(* PLC project HydMotion Functions library, Porcheson Hydraulic Motion 0.0 *)
(* stored: creationDateTime 2023-02-10T00:00:00, modificationDateTime 2026-02-10T00:00:00 *)

TYPE HYD_AxisMotion : STRUCT
  SEGMENTTAG : USINT;
  SEGMENTTYPE : USINT;
  PLANNER : USINT;
  MODE : USINT;
  ENDCONDITION : USINT;
  DIRECTION : USINT;
  SETPOSITION : REAL;
  SETVELOCITY : REAL;  (* 仅在速度/流量控制模式下使用，表示目标速度； *)
  SETFLOW : REAL;  (* 仅在速度/流量控制模式下使用，表示目标流量；在位置控制模式下忽略 *)
  SETPRESSURE : REAL;
  ACCELERATION : REAL;
  DECELERATION : REAL;
  DURATION : REAL;
  PRESSURERAMPRATE : REAL;
  ACTPOSITION : REAL;
  ACTVELOCITY : REAL;
  ACTFLOW : REAL;
  ACTPRESSURE : REAL;
  TIMESTAMP : REAL;
END_STRUCT;
END_TYPE

FUNCTION_BLOCK HYD_MoveProfile
  VAR_INPUT
    AXISID : SINT;
    EXECUTE : BOOL;
    MOTION : HYD_AxisMotion;
    BUFFERMODE : INT;
  END_VAR
  VAR_OUTPUT
    DONE : BOOL;
    BUSY : BOOL;
    ACTIVE : BOOL;
    COMMANDABORTED : BOOL;
    ERROR : BOOL;
    ERRORID : WORD;
  END_VAR
  VAR
    Execute0 : BOOL;
    Done0 : BOOL;
    Active0 : BOOL;
    _PENDING : BOOL;
    _EXEC_ID : WORD;
  END_VAR

 {{ extern void __mcl_cmd_MoveProfile(HYD_MOVEPROFILE *data__);	__mcl_cmd_MoveProfile(data__);	 }}			
END_FUNCTION_BLOCK

FUNCTION_BLOCK HYD_LoadProfile
  VAR_INPUT
    AXISID : SINT;
    EXECUTE : BOOL;
    MOTION : HYD_AxisMotion;
  END_VAR
  VAR_OUTPUT
    DONE : BOOL;
    BUSY : BOOL;
    ERROR : BOOL;
    ERRORID : WORD;
  END_VAR
  VAR
    Execute0 : BOOL;
    Done0 : BOOL;
  END_VAR

						{{ extern void __mcl_cmd_LoadProfile(HYD_LOADPROFILE *data__);	__mcl_cmd_LoadProfile(data__);	 }}	
					
END_FUNCTION_BLOCK

FUNCTION_BLOCK HYD_Stop
  VAR_INPUT
    AXISID : SINT;
    EXECUTE : BOOL;
    DECELERATION : REAL;
  END_VAR
  VAR_OUTPUT
    DONE : BOOL;
    BUSY : BOOL;
    COMMANDABORTED : BOOL;
    ERROR : BOOL;
    ERRORID : WORD;
  END_VAR
  VAR
    Execute0 : BOOL;
    Done0 : BOOL;
    Active0 : BOOL;
    _PENDING : BOOL;
  END_VAR

						{{ extern void __mcl_cmd_Stop(HYD_STOP *data__);	__mcl_cmd_Stop(data__);	 }}	
					
END_FUNCTION_BLOCK

FUNCTION_BLOCK HYD_Hold
  VAR_INPUT
    AXISID : SINT;
    EXECUTE : BOOL;
  END_VAR
  VAR_OUTPUT
    DONE : BOOL;
    BUSY : BOOL;
    ERROR : BOOL;
    ERRORID : WORD;
  END_VAR
  VAR
    EXECUTE0 : BOOL;
    DONE0 : BOOL;
    _PENDING : BOOL;
  END_VAR

{{ extern void __mcl_cmd_Hold(HYD_HOLD*); __mcl_cmd_Hold(data__); }} 
END_FUNCTION_BLOCK

FUNCTION_BLOCK HYD_Resume
  VAR_INPUT
    AXISID : SINT;
    EXECUTE : BOOL;
  END_VAR
  VAR_OUTPUT
    DONE : BOOL;
    BUSY : BOOL;
    ERROR : BOOL;
    ERRORID : WORD;
  END_VAR
  VAR
    EXECUTE0 : BOOL;
    DONE0 : BOOL;
    _PENDING : BOOL;
  END_VAR

{{ extern void __mcl_cmd_Resume(HYD_RESUME*); __mcl_cmd_Resume(data__); }} 
END_FUNCTION_BLOCK

(* This Function Block commands a controlled motion to a specified absolute position. *)
FUNCTION_BLOCK HYD_MoveAbsolute
  VAR_INPUT
    AXISID : SINT;
    EXECUTE : BOOL;
    CONTINUOUSUPDATE : BOOL;
    POSITION : REAL;
    VELOCITY : REAL;
    ACCELERATION : REAL;
    DECELERATION : REAL;
    JERK : REAL;
    DIRECTION : SINT;
    BUFFERMODE : INT;
  END_VAR
  VAR_OUTPUT
    DONE : BOOL;
    BUSY : BOOL;
    ACTIVE : BOOL;
    COMMANDABORTED : BOOL;
    ERROR : BOOL;
    ERRORID : WORD;
  END_VAR
  VAR
    EXECUTE0 : BOOL;
    DONE0 : BOOL;
    ACTIVE0 : BOOL;
    _PENDING : BOOL;
    _EXEC_ID : WORD;
  END_VAR

						{{ extern void __mcl_cmd_MoveAbsolute(HYD_MOVEABSOLUTE*); __mcl_cmd_MoveAbsolute(data__); }}	
					
END_FUNCTION_BLOCK

FUNCTION_BLOCK HYD_MoveContinuousAbsolute
  VAR_INPUT
    AXISID : SINT;
    EXECUTE : BOOL;
    POSITION : REAL;
    VELOCITY : REAL;
    ENDVELOCITY : REAL;
    ENDVELOCITYDIRECTION : SINT;
    ACCELERATION : REAL;
    DECELERATION : REAL;
    JERK : REAL;
    DIRECTION : SINT;
    ADAPTENDVELTOAVOIDOVERSHOOT : BOOL;
    PRESSURELIMIT : REAL;
  END_VAR
  VAR_OUTPUT
    INENDVELOCITY : BOOL;
    POSITIONREACHED : BOOL;
    BUSY : BOOL;
    COMMANDABORTED : BOOL;
    ERROR : BOOL;
    ERRORID : WORD;
  END_VAR
  VAR
    EXECUTE0 : BOOL;
    INENDVELOCITY0 : BOOL;
    POSITIONREACHED0 : BOOL;
    _PENDING : BOOL;
    _EXEC_ID : WORD;
  END_VAR

{{ extern void __mcl_cmd_MoveContinuousAbsolute(HYD_MOVECONTINUOUSABSOLUTE*); __mcl_cmd_MoveContinuousAbsolute(data__); }} 
END_FUNCTION_BLOCK

(* This Function Block commands a never ending controlled motion at a specified velocity. *)
FUNCTION_BLOCK HYD_MoveVelocity
  VAR_INPUT
    AXISID : SINT;
    EXECUTE : BOOL;
    CONTINUOUSUPDATE : BOOL;
    VELOCITY : REAL;
    ACCELERATION : REAL;
    DECELERATION : REAL;
    JERK : REAL;
    DIRECTION : SINT;
    BUFFERMODE : INT;
    PRESSURELIMIT : REAL;
  END_VAR
  VAR_OUTPUT
    INVELOCITY : BOOL;
    BUSY : BOOL;
    ACTIVE : BOOL;
    COMMANDABORTED : BOOL;
    ERROR : BOOL;
    ERRORID : WORD;
  END_VAR
  VAR
    EXECUTE0 : BOOL;
    INVELOCITY0 : BOOL;
    ACTIVE0 : BOOL;
    _PENDING : BOOL;
    _EXEC_ID : WORD;
  END_VAR

{{ extern void __mcl_cmd_MoveVelocity(HYD_MOVEVELOCITY*); __mcl_cmd_MoveVelocity(data__); }} 
END_FUNCTION_BLOCK

(* This Function Block makes the transition from the state ‘ErrorStop’ to ‘Disabled’ by resetting all internal axis-related errors *)
FUNCTION_BLOCK HYD_Reset
  VAR_INPUT
    AXISID : SINT;
    EXECUTE : BOOL;
  END_VAR
  VAR_OUTPUT
    DONE : BOOL;
    BUSY : BOOL;
    ERROR : BOOL;
    ERRORID : WORD;
  END_VAR
  VAR
    EXECUTE0 : BOOL;
    DONE0 : BOOL;
  END_VAR

{{ extern void __mcl_cmd_Reset(HYD_RESET*); __mcl_cmd_Reset(data__); }} 
END_FUNCTION_BLOCK

(* This Function Block commands pressure closed control. FLOWLIMITPERCENT is the pressure-segment flow cap as a percentage of 20 L/min; valid range is (0,100], default 100. *)
FUNCTION_BLOCK HYD_PressureHandle
  VAR_INPUT
    AXISID : SINT;
    EXECUTE : BOOL;
    CONTINUOUSUPDATE : BOOL;
    PRESSURE : REAL;
    PRESSURERAMPRATE : REAL;
    DURATION : REAL;
    FLOWLIMITPERCENT : REAL := 100;
    BUFFERMODE : INT;
  END_VAR
  VAR_OUTPUT
    INPRESSURE : BOOL;
    DONE : BOOL;
    BUSY : BOOL;
    ACTIVE : BOOL;
    COMMANDABORTED : BOOL;
    ERROR : BOOL;
    ERRORID : WORD;
  END_VAR
  VAR
    EXECUTE0 : BOOL;
    INPRESSURE0 : BOOL;
    ACTIVE0 : BOOL;
    _PENDING : BOOL;
    _EXEC_ID : WORD;
  END_VAR

{{ extern void __mcl_cmd_PressureHandle(HYD_PRESSUREHANDLE*); __mcl_cmd_PressureHandle(data__); }} 
END_FUNCTION_BLOCK

(* This allocates a simulation Axis, for testing.One axis per instanciated FB. *)
FUNCTION_BLOCK HYD_CreateMotion
  VAR_INPUT
    USE_RECIPE : BOOL := 0;
    FLOW_TO_PUMPSPEED : REAL := 20.0;
    PUMPSPEED_LIMIT : REAL := 1800.0;
    USE_SIMULATION : BOOL := 0;
    MECHANISM_TYPE : SINT := 0;
  END_VAR
  VAR_OUTPUT
    AXISID : SINT;
    DONE : BOOL;
    BUSY : BOOL;
    ERROR : BOOL;
    ERRORID : WORD;
  END_VAR
  VAR
    DONE0 : BOOL;
    _RESERVED_AXIS : SINT;
    _RESERVED_SLOT : USINT;
    _VALIDATION_TOKEN : USINT;
    _CREATE_ACTIVE : BOOL;
    _FRAMEWORK_GENERATION : WORD;
  END_VAR

						{{ extern void __mcl_cmd_CreateMotion(HYD_CREATEMOTION*); __mcl_cmd_CreateMotion(data__); }} 
					
END_FUNCTION_BLOCK

(* Atomically validates and commits five-point toggle geometry. *)
FUNCTION_BLOCK HYD_ConfigureToggleMechanism
  VAR_INPUT
    AXISID : SINT;
    EXECUTE : BOOL;
    LR : LREAL;
    LF : LREAL;
    LPF : LREAL;
    LPK : LREAL;
    LD : LREAL;
    HF : LREAL;
    HM : LREAL;
    DC : LREAL;
    SM : LREAL;
    XHANDOFF : LREAL;
    SIGMA_K : SINT;
    SIGN_B : SINT;
    TAU_S : SINT;
    SIGMA_C : SINT := -1;
  END_VAR
  VAR_OUTPUT
    DONE : BOOL;
    BUSY : BOOL;
    ERROR : BOOL;
    ERRORID : WORD;
    CONFIG_VERSION : WORD;
  END_VAR
  VAR
    EXECUTE0 : BOOL;
    VALIDATION_TOKEN : USINT;
    ACTIVE : BOOL;
    CONFIG_AXIS : SINT;
    _FRAMEWORK_GENERATION : WORD;
  END_VAR

{{ extern void __mcl_cmd_ConfigureToggleMechanism(HYD_CONFIGURETOGGLEMECHANISM*); __mcl_cmd_ConfigureToggleMechanism(data__); }} 
END_FUNCTION_BLOCK

(* Reads the committed five-point toggle geometry and safe envelope. *)
FUNCTION_BLOCK HYD_ReadToggleMechanism
  VAR_INPUT
    AXISID : SINT;
    ENABLE : BOOL;
  END_VAR
  VAR_OUTPUT
    VALID : BOOL;
    USING_DEFAULTS : BOOL;
    LR : LREAL;
    LF : LREAL;
    LPF : LREAL;
    LPK : LREAL;
    LD : LREAL;
    HF : LREAL;
    HM : LREAL;
    DC : LREAL;
    SM : LREAL;
    XHANDOFF : LREAL;
    SIGMA_K : SINT;
    SIGN_B : SINT;
    TAU_S : SINT;
    SIGMA_C : SINT;
    CONFIG_VERSION : WORD;
    X_GEOMETRY_MIN : LREAL;
    X_HANDOFF_EFFECTIVE : LREAL;
    XS_MIN : LREAL;
    XS_MAX : LREAL;
    K_MIN : LREAL;
    K_MAX : LREAL;
    ERROR : BOOL;
    ERRORID : WORD;
  END_VAR

{{ extern void __mcl_cmd_ReadToggleMechanism(HYD_READTOGGLEMECHANISM*); __mcl_cmd_ReadToggleMechanism(data__); }} 
END_FUNCTION_BLOCK

(* set feedback to motion. *)
FUNCTION_BLOCK HYD_SetAxisFeedback
  VAR_INPUT
    AXISID : SINT;
    ENABLE : BOOL;
    ACT_POSITION : REAL;
    ACT_VELOCITY : REAL;
    ACT_FLOW : REAL;
    ACT_PRESSURE : REAL;
    TIMESTAMP : REAL;
  END_VAR
  VAR_OUTPUT
    DONE : BOOL;
    BUSY : BOOL;
    ERROR : BOOL;
    ERRORID : WORD;
  END_VAR
  VAR
    DONE0 : BOOL;
  END_VAR

						{{ extern void __mcl_cmd_SetAxisFeedback(HYD_SETAXISFEEDBACK*); __mcl_cmd_SetAxisFeedback(data__); }} 
					
END_FUNCTION_BLOCK

(* write shared system-level pump feedback; one pump serves multiple axes. *)
FUNCTION_BLOCK HYD_SetPumpFeedback
  VAR_INPUT
    ENABLE : BOOL;
    PUMP_SPEED_RPM : REAL;
    PUMP_ANGLE_DEG : REAL;
    PUMP_TORQUE_PCT_TN : REAL;
    TIMESTAMP : REAL;
  END_VAR
  VAR_OUTPUT
    DONE : BOOL;
    BUSY : BOOL;
    ERROR : BOOL;
    ERRORID : WORD;
  END_VAR

{{ extern void __mcl_cmd_SetPumpFeedback(HYD_SETPUMPFEEDBACK*); __mcl_cmd_SetPumpFeedback(data__); }} 
END_FUNCTION_BLOCK

(* get only one pump speed command from motion. *)
FUNCTION_BLOCK HYD_GetPumpRequest
  VAR_INPUT
    ENABLE : BOOL;
    STRATEGY : SINT;
    ALLOW_NEGATIVE : BOOL;
  END_VAR
  VAR_OUTPUT
    PUMPSPEED : REAL;
    CONFLICT : BOOL;
    BUSY : BOOL;
    DONE : BOOL;
    ERROR : BOOL;
    ERRORID : WORD;
  END_VAR
  VAR
    DONE0 : BOOL;
  END_VAR

						{{ extern void __mcl_cmd_GetPumpRequest(HYD_GETPUMPREQUEST*); __mcl_cmd_GetPumpRequest(data__); }} 
					
END_FUNCTION_BLOCK

(* get axis status from motion. *)
FUNCTION_BLOCK HYD_ReadStatus
  VAR_INPUT
    AXISID : SINT;
    ENABLE : BOOL;
  END_VAR
  VAR_OUTPUT
    VALID : BOOL;
    BUSY : BOOL;
    ERROR : BOOL;
    ERRORID : WORD;
    STATE : UINT;
    PRESSURECONTROLLERAPPLIED : INT;
    MECHANISMTYPE : SINT;
    ACTUATORDIRECTION : SINT;
    ACTUATORPOSITION : REAL;
    ACTUATORVELOCITYCOMMAND : REAL;
    VELOCITYRATIO : REAL;
    MECHANISMCONFIGVERSION : WORD;
    REQUESTEDFLOW : REAL;
    MAXFLOW : REAL;
    MAXTEMPLATEVELOCITY : REAL;
    EFFECTIVECYLINDERGAIN : REAL;
    FLOWLIMITACTIVE : BOOL;
    PUMPSPEEDLIMITACTIVE : BOOL;
    PRESSURELIMITACTIVE : BOOL;
    SOFTLIMITACTIVE : BOOL;
    DERATED : BOOL;
  END_VAR

						{{ extern void __mcl_cmd_ReadStatus(HYD_READSTATUS*); __mcl_cmd_ReadStatus(data__); }} 
					
END_FUNCTION_BLOCK

(* get axis error from motion. *)
FUNCTION_BLOCK HYD_ReadError
  VAR_INPUT
    AXISID : SINT;
    ENABLE : BOOL;
  END_VAR
  VAR_OUTPUT
    VALID : BOOL;
    BUSY : BOOL;
    ERROR : BOOL;
    ERRORID : WORD;
  END_VAR

						{{ extern void __mcl_cmd_ReadError(HYD_READERROR*); __mcl_cmd_ReadError(data__); }} 
					
END_FUNCTION_BLOCK

(* get axis simfeedback from motion. *)
FUNCTION_BLOCK HYD_ReadSimFeedback
  VAR_INPUT
    AXISID : SINT;
    ENABLE : BOOL;
  END_VAR
  VAR_OUTPUT
    VALID : BOOL;
    BUSY : BOOL;
    ERROR : BOOL;
    ERRORID : WORD;
    POSITION : REAL;
    VELOCITY : REAL;
    FLOW : REAL;
    PRESSURE : REAL;
  END_VAR

						{{ extern void __mcl_cmd_ReadSimFeedback(HYD_READSIMFEEDBACK*); __mcl_cmd_ReadSimFeedback(data__); }} 
					
END_FUNCTION_BLOCK

FUNCTION_BLOCK HYD_ReadParameter
  VAR_INPUT
    AXISID : SINT;
    ENABLE : BOOL;
    PARAMETERNUMBER : INT;
  END_VAR
  VAR_OUTPUT
    VALID : BOOL;
    BUSY : BOOL;
    ERROR : BOOL;
    ERRORID : WORD;
    VALUE : LREAL;
  END_VAR
  VAR
    ENABLE0 : BOOL;
  END_VAR

{{ extern void __mcl_cmd_ReadParameter(HYD_READPARAMETER*); __mcl_cmd_ReadParameter(data__); }}
END_FUNCTION_BLOCK

FUNCTION_BLOCK HYD_WriteParameter
  VAR_INPUT
    AXISID : SINT;
    EXECUTE : BOOL;
    PARAMETERNUMBER : INT;
    VALUE : LREAL;
  END_VAR
  VAR_OUTPUT
    DONE : BOOL;
    BUSY : BOOL;
    ERROR : BOOL;
    ERRORID : WORD;
  END_VAR
  VAR
    EXECUTE0 : BOOL;
    DONE0 : BOOL;
  END_VAR

{{ extern void __mcl_cmd_WriteParameter(HYD_WRITEPARAMETER*); __mcl_cmd_WriteParameter(data__); }}
END_FUNCTION_BLOCK

FUNCTION_BLOCK HYD_ReadBoolParameter
  VAR_INPUT
    AXISID : SINT;
    ENABLE : BOOL;
    PARAMETERNUMBER : INT;
  END_VAR
  VAR_OUTPUT
    VALID : BOOL;
    BUSY : BOOL;
    ERROR : BOOL;
    ERRORID : WORD;
    VALUE : BOOL;
  END_VAR
  VAR
    ENABLE0 : BOOL;
  END_VAR

{{ extern void __mcl_cmd_ReadBoolParameter(HYD_READBOOLPARAMETER*); __mcl_cmd_ReadBoolParameter(data__); }}
END_FUNCTION_BLOCK

FUNCTION_BLOCK HYD_WriteBoolParameter
  VAR_INPUT
    AXISID : SINT;
    EXECUTE : BOOL;
    PARAMETERNUMBER : INT;
    VALUE : BOOL;
  END_VAR
  VAR_OUTPUT
    DONE : BOOL;
    BUSY : BOOL;
    ERROR : BOOL;
    ERRORID : WORD;
  END_VAR
  VAR
    EXECUTE0 : BOOL;
    DONE0 : BOOL;
  END_VAR

{{ extern void __mcl_cmd_WriteBoolParameter(HYD_WRITEBOOLPARAMETER*); __mcl_cmd_WriteBoolParameter(data__); }}
END_FUNCTION_BLOCK
